// TwinCAT 3 PLC project Array_Flexible
// ProgramVersion: 3.1.4024.0
// libraries:
//   Tc2_Standard, * (Beckhoff Automation GmbH)
//   Tc2_System, * (Beckhoff Automation GmbH)
//   Tc3_Module, * (Beckhoff Automation GmbH)
// project tree:
//   / PlcTask.TcTTO
//   POUs/ FSum.TcPOU, MAIN.TcPOU
// real-time tasks:
//   TASK PlcTask: cycle T#10ms, priority 20, ADS port 350

CONFIGURATION Array_Flexible
    RESOURCE PLC ON TwinCAT3
        TASK PlcTask(INTERVAL := T#10ms, PRIORITY := 20);
        PROGRAM MAIN WITH PlcTask : MAIN;
    END_RESOURCE
END_CONFIGURATION

// ---- POUs/MAIN.TcPOU
PROGRAM MAIN
VAR
	aArr1 	: ARRAY[0..10] OF INT 	:= [1,1,1,1,1,1,1,1,1,1,1]; 
	aArr2  	: ARRAY[0..5] OF INT 	:= [2,2,2,2,2,2];
	aArr3  	: ARRAY[0..1] OF INT 	:= [10,10];
	sum1	: DINT;
	sum2	: DINT;
	sum3	: DINT;
END_VAR


sum1 := Fsum(aData := aArr1);
sum2 := Fsum(aData := aArr2);
sum3 := Fsum(aData := aArr3);

END_PROGRAM

// ---- POUs/FSum.TcPOU
FUNCTION FSum : dint
VAR_IN_OUT
    aData     : ARRAY [*] OF INT;
END_VAR
VAR
    i, nSum   : DINT;
END_VAR

nSum := 0;
 
FOR i := LOWER_BOUND(aData,1) TO UPPER_BOUND(aData,1) DO
    nSum := nSum + aData[i];
END_FOR;

FSum := nSum;

END_FUNCTION
